Xinje XDPPro project, PLC1: XD5-48T6 (software 3.5.3 2018-11-19)

PROGRAM Ladder

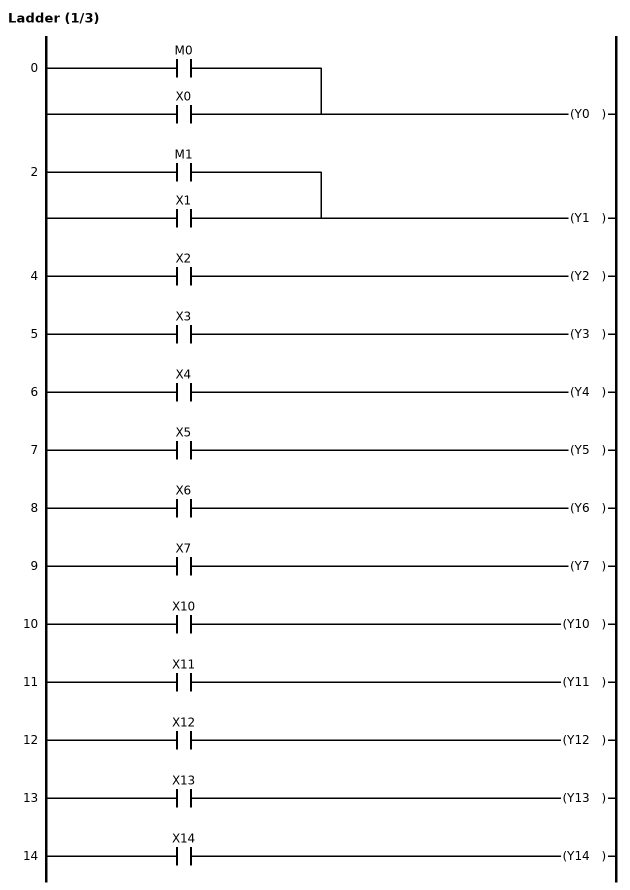
LD     M0
OR     X0
OUT    Y0
LD     M1
OR     X1
OUT    Y1
LD     X2
OUT    Y2
LD     X3
OUT    Y3
LD     X4
OUT    Y4
LD     X5
OUT    Y5
LD     X6
OUT    Y6
LD     X7
OUT    Y7
LD     X10
OUT    Y10
LD     X11
OUT    Y11
LD     X12
OUT    Y12
LD     X13
OUT    Y13
LD     X14
OUT    Y14

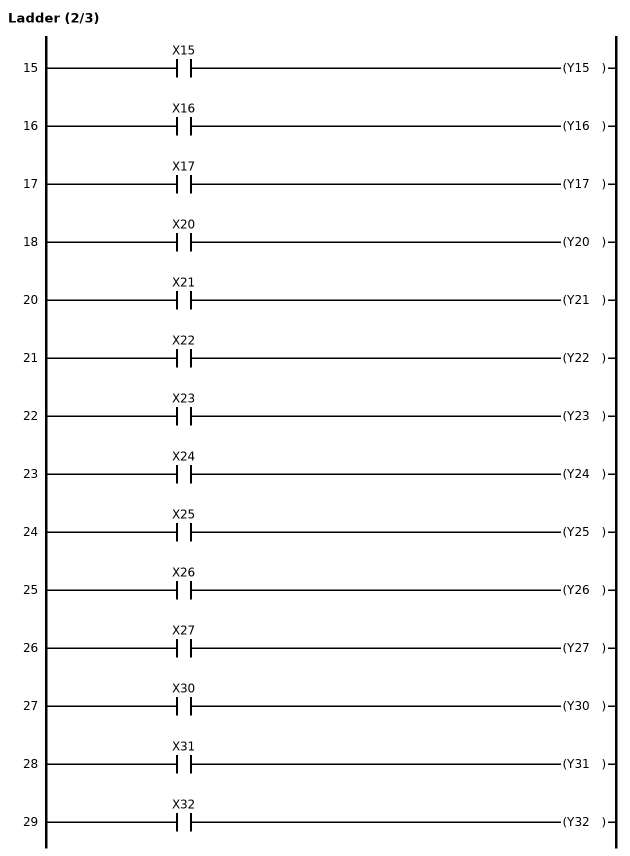
LD     X15
OUT    Y15
LD     X16
OUT    Y16
LD     X17
OUT    Y17
LD     X20
OUT    Y20
LD     X21
OUT    Y21
LD     X22
OUT    Y22
LD     X23
OUT    Y23
LD     X24
OUT    Y24
LD     X25
OUT    Y25
LD     X26
OUT    Y26
LD     X27
OUT    Y27
LD     X30
OUT    Y30
LD     X31
OUT    Y31
LD     X32
OUT    Y32

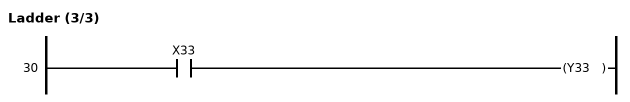
LD     X33
OUT    Y33